TYPE ST_CSV_Record :
STRUCT
sName 	: T_MaxString 	:= '';
	nNumber	: UDINT 		:= 0;
	fPos	: LREAL 		:= 0.0;
	bOP		: BOOL 			:= FALSE;
	sDesc	: STRING(40)	:= '';
	data	: ARRAY[0..7] OF BYTE;
END_STRUCT
END_TYPE

(* stored: Version 1.1.0.1, ProductVersion 3.1.4024.12
   DUT ST_CSV_Record: Id {54243cf1-d582-4bd4-be96-d59efd381c73} *)
